(* IEC 61131-3 sources: RL_MAR/experiments/comparison/llm4plc/results/Qwen-Qwen3.5-9B_20260506_150728/20260506_162616, 4 files *)

(* ---- generated_code_iteration_0.st ---- *)
START_ST
FUNCTION_BLOCK FB_MergeBytes
VAR_INPUT
    byteArray : ARRAY[1..20] OF DINT; (* Byte array to be merged *)
END_VAR
VAR_OUTPUT
    dwordArray : ARRAY[1..10] OF DINT; (* Merged double word array *)
    mergeDwordNum : DINT; (* Actual number of merged double words *)
END_VAR
VAR
    k : INT; (* Loop counter for double words *)
    b1, b2, b3, b4 : DINT; (* Temporary byte holders *)
    tempDword : DINT; (* Accumulated result *)
    maxMerges : DINT; (* Potential merges based on input size *)
    limit : DINT; (* Actual merges based on input and output size *)
    BYTE_ARRAY_SIZE : DINT := 20;
    DWORD_ARRAY_SIZE : DINT := 10;
END_VAR
VAR CONSTANT
    SHIFT_8 : DINT := 256;
    SHIFT_16 : DINT := 65536;
    SHIFT_24 : DINT := 16777216;
END_VAR

BEGIN
    (* STATE 0: INITIALIZE *)
    mergeDwordNum := 0;
    FOR i := 1 TO DWORD_ARRAY_SIZE DO
        dwordArray[i] := 0;
    END_FOR;

    (* STATE 1: CALCULATE LIMITS *)
    maxMerges := BYTE_ARRAY_SIZE DIV 4;
    IF maxMerges > DWORD_ARRAY_SIZE THEN
        limit := DWORD_ARRAY_SIZE;
    ELSE
        limit := maxMerges;
    END_IF;

    (* STATE 2: MERGE AND STORE LOOP *)
    FOR k := 0 TO limit - 1 DO
        (* Check if 4 bytes exist at index k*4 *)
        IF (k * 4 + 4) <= BYTE_ARRAY_SIZE THEN
            (* Extract 4 bytes: byteArray[k*4+1] to byteArray[k*4+4] *)
            b1 := byteArray[(k * 4) + 1];
            b2 := byteArray[(k * 4) + 2];
            b3 := byteArray[(k * 4) + 3];
            b4 := byteArray[(k * 4) + 4];

            (* Construct tempDword (Little Endian: Byte1=LSB, Byte4=MSB) *)
            tempDword := b1 + (b2 * SHIFT_8) + (b3 * SHIFT_16) + (b4 * SHIFT_24);

            (* Store result *)
            dwordArray[k + 1] := tempDword;

            (* Increment counter *)
            mergeDwordNum := mergeDwordNum + 1;
        ELSE
            (* Insufficient bytes, exit loop *)
            EXIT;
        END_IF;
    END_FOR;

    (* STATE 3: FINALIZE - Counter already updated inside loop *)
END_FUNCTION_BLOCK
END_ST

(* ---- generated_code_iteration_1.st ---- *)
START_REASON
The validation feedback indicates a CODESYS compiler error: "发现非预期的记号'limit'" (Unexpected token 'limit').

Analysis of the error:
1.  **Variable Declaration Conflict**: In the `VAR` section, I declared a variable named `limit`. However, in CODESYS Structured Text, `limit` is often a reserved keyword or a standard library function name (e.g., used in `LIMIT` functions or specific STL contexts), or simply a naming convention that the compiler flags as unexpected in this specific context if not strictly adhered to.
2.  **Variable Initialization**: The variable `limit` was declared but not initialized with a default value or assigned before use in a way that might trigger scope issues if the compiler expects a constant or a specific type.
3.  **Best Practice**: To avoid ambiguity and potential reserved word conflicts in CODESYS, it is best to rename variables that look like keywords or standard functions. I will rename `limit` to `maxMergesCount` or similar.
4.  **Logic Check**: The logic for merging bytes into double words (DINT) is sound, but the variable naming is the primary blocker. I will also ensure all variables are properly typed and initialized.

Plan:
1.  Rename the variable `limit` to `mergeCount` to avoid the "unexpected token" error.
2.  Ensure the `VAR` section is clean and follows strict ST rules.
3.  Maintain the `FUNCTION_BLOCK` structure.
4.  Ensure `END_VAR` is used correctly to close sections.
END_REASON

START_ST
FUNCTION_BLOCK FB_MergeBytes
VAR_INPUT
    byteArray : ARRAY[1..20] OF DINT; (* Byte array to be merged *)
END_VAR
VAR_OUTPUT
    dwordArray : ARRAY[1..10] OF DINT; (* Merged double word array *)
    mergeDwordNum : DINT; (* Actual number of merged double words *)
END_VAR
VAR
    k : INT; (* Loop counter for double words *)
    i : INT; (* Loop counter for initialization *)
    b1, b2, b3, b4 : DINT; (* Temporary byte holders *)
    tempDword : DINT; (* Accumulated result *)
    maxMerges : DINT; (* Potential merges based on input size *)
    mergeCount : DINT; (* Actual merges based on input and output size - Renamed from 'limit' *)
    BYTE_ARRAY_SIZE : DINT := 20;
    DWORD_ARRAY_SIZE : DINT := 10;
END_VAR
VAR CONSTANT
    SHIFT_8 : DINT := 256;
    SHIFT_16 : DINT := 65536;
    SHIFT_24 : DINT := 16777216;
END_VAR

BEGIN
    (* STATE 0: INITIALIZE *)
    mergeDwordNum := 0;
    FOR i := 1 TO DWORD_ARRAY_SIZE DO
        dwordArray[i] := 0;
    END_FOR;

    (* STATE 1: CALCULATE LIMITS *)
    maxMerges := BYTE_ARRAY_SIZE DIV 4;
    IF maxMerges > DWORD_ARRAY_SIZE THEN
        mergeCount := DWORD_ARRAY_SIZE;
    ELSE
        mergeCount := maxMerges;
    END_IF;

    (* STATE 2: MERGE AND STORE LOOP *)
    FOR k := 0 TO mergeCount - 1 DO
        (* Check if 4 bytes exist at index k*4 *)
        IF (k * 4 + 4) <= BYTE_ARRAY_SIZE THEN
            (* Extract 4 bytes: byteArray[k*4+1] to byteArray[k*4+4] *)
            b1 := byteArray[(k * 4) + 1];
            b2 := byteArray[(k * 4) + 2];
            b3 := byteArray[(k * 4) + 3];
            b4 := byteArray[(k * 4) + 4];

            (* Construct tempDword (Little Endian: Byte1=LSB, Byte4=MSB) *)
            tempDword := b1 + (b2 * SHIFT_8) + (b3 * SHIFT_16) + (b4 * SHIFT_24);

            (* Store result *)
            dwordArray[k + 1] := tempDword;

            (* Increment counter *)
            mergeDwordNum := mergeDwordNum + 1;
        ELSE
            (* Insufficient bytes, exit loop *)
            EXIT;
        END_IF;
    END_FOR;

    (* STATE 3: FINALIZE - Counter already updated inside loop *)
END_FUNCTION_BLOCK
END_ST

(* ---- generated_code_iteration_2.st ---- *)
START_REASON
The previous code failed due to an encoding issue (illegal multibyte sequence 0xa2). This typically happens when special characters (like Chinese comments or invisible formatting characters) are present in the source code, which the CODESYS compiler cannot parse in the expected ASCII/UTF-8 environment.

Additionally, while the logic was improved by renaming the variable, the comment syntax `(* ... *)` is correct, but the content might have contained hidden non-ASCII characters. To ensure robustness, I will:
1.  Remove all comments to eliminate any potential encoding artifacts.
2.  Ensure all variable names and keywords are strictly ASCII.
3.  Maintain the `FUNCTION_BLOCK` structure and correct `END_VAR` usage.
4.  Keep the logic intact: merging 4 DINTs into 1 DINT (interpreted as bytes here based on the shift logic, though the type is DINT, the math implies byte-level shifting). The logic calculates how many 4-byte chunks fit and merges them.

The core fix is sanitizing the text to pure ASCII to resolve the "illegal multibyte sequence" error.
END_REASON

START_ST
FUNCTION_BLOCK FB_MergeBytes
VAR_INPUT
    byteArray : ARRAY[1..20] OF DINT;
END_VAR
VAR_OUTPUT
    dwordArray : ARRAY[1..10] OF DINT;
    mergeDwordNum : DINT;
END_VAR
VAR
    k : INT;
    i : INT;
    b1, b2, b3, b4 : DINT;
    tempDword : DINT;
    maxMerges : DINT;
    mergeCount : DINT;
    BYTE_ARRAY_SIZE : DINT := 20;
    DWORD_ARRAY_SIZE : DINT := 10;
END_VAR
VAR CONSTANT
    SHIFT_8 : DINT := 256;
    SHIFT_16 : DINT := 65536;
    SHIFT_24 : DINT := 16777216;
END_VAR

BEGIN
    mergeDwordNum := 0;
    FOR i := 1 TO DWORD_ARRAY_SIZE DO
        dwordArray[i] := 0;
    END_FOR;

    maxMerges := BYTE_ARRAY_SIZE DIV 4;
    IF maxMerges > DWORD_ARRAY_SIZE THEN
        mergeCount := DWORD_ARRAY_SIZE;
    ELSE
        mergeCount := maxMerges;
    END_IF;

    FOR k := 0 TO mergeCount - 1 DO
        IF (k * 4 + 4) <= BYTE_ARRAY_SIZE THEN
            b1 := byteArray[(k * 4) + 1];
            b2 := byteArray[(k * 4) + 2];
            b3 := byteArray[(k * 4) + 3];
            b4 := byteArray[(k * 4) + 4];

            tempDword := b1 + (b2 * SHIFT_8) + (b3 * SHIFT_16) + (b4 * SHIFT_24);

            dwordArray[k + 1] := tempDword;
            mergeDwordNum := mergeDwordNum + 1;
        ELSE
            EXIT;
        END_IF;
    END_FOR;
END_FUNCTION_BLOCK
END_ST

(* ---- generated_code_iteration_3.st ---- *)
START_REASON
The previous code failed because the variable name `mergeDwordNum` contains a Chinese character ('字', meaning 'character' or 'word'). The CODESYS compiler strictly requires all variable names to be ASCII characters only. The error message "应该用';' 替换'mergeDwordNum'" translates to "Should replace 'mergeDwordNum' with ';'", which is a cryptic way of indicating that the non-ASCII character in the name is invalid and needs to be replaced (effectively removing the variable or renaming it to valid ASCII).

To fix this:
1. Rename `mergeDwordNum` to `mergeDwordCount` (pure ASCII).
2. Ensure all other variable names are also strictly ASCII (e.g., `byteArray`, `dwordArray`, `tempDword`, etc., are already compliant).
3. Maintain the `FUNCTION_BLOCK` structure and `END_VAR` usage.
4. Keep the logic intact.
END_REASON

START_ST
FUNCTION_BLOCK FB_MergeBytes
VAR_INPUT
    byteArray : ARRAY[1..20] OF DINT;
END_VAR
VAR_OUTPUT
    dwordArray : ARRAY[1..10] OF DINT;
    mergeDwordCount : DINT;
END_VAR
VAR
    k : INT;
    i : INT;
    b1, b2, b3, b4 : DINT;
    tempDword : DINT;
    maxMerges : DINT;
    mergeCount : DINT;
    BYTE_ARRAY_SIZE : DINT := 20;
    DWORD_ARRAY_SIZE : DINT := 10;
END_VAR
VAR CONSTANT
    SHIFT_8 : DINT := 256;
    SHIFT_16 : DINT := 65536;
    SHIFT_24 : DINT := 16777216;
END_VAR

BEGIN
    mergeDwordCount := 0;
    FOR i := 1 TO DWORD_ARRAY_SIZE DO
        dwordArray[i] := 0;
    END_FOR;

    maxMerges := BYTE_ARRAY_SIZE DIV 4;
    IF maxMerges > DWORD_ARRAY_SIZE THEN
        mergeCount := DWORD_ARRAY_SIZE;
    ELSE
        mergeCount := maxMerges;
    END_IF;

    FOR k := 0 TO mergeCount - 1 DO
        IF (k * 4 + 4) <= BYTE_ARRAY_SIZE THEN
            b1 := byteArray[(k * 4) + 1];
            b2 := byteArray[(k * 4) + 2];
            b3 := byteArray[(k * 4) + 3];
            b4 := byteArray[(k * 4) + 4];

            tempDword := b1 + (b2 * SHIFT_8) + (b3 * SHIFT_16) + (b4 * SHIFT_24);

            dwordArray[k + 1] := tempDword;
            mergeDwordCount := mergeDwordCount + 1;
        ELSE
            EXIT;
        END_IF;
    END_FOR;
END_FUNCTION_BLOCK
END_ST
